FUNCTION_BLOCK OUT_ANY_TEST (* Data output to TextField *)
  (* Standard: 61499-1; Classification: GUI *)
  (* Version 0.3, 2009-02-28, JHC, Holobloc Inc, Updated service sequences. *)
  (* Version 0.2, 2009-02-23, JHC, Holobloc Inc, Updated compilers. *)
  (* Version 0.1, 2002-05-03, JHC, Rockwell Automation, Made QI IV=true. *)
  (* Version 0.0, 2001-05-31, JHC, Rockwell Automation *)
  (* Compiler header: package fb.rt.hmi; *)
  (* Compiler Java Sun JDK 1.6.0 *)
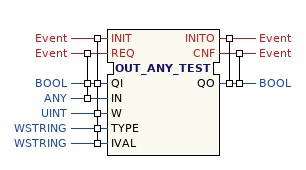
  EVENT_INPUT
    INIT WITH QI, W, TYPE, IVAL; (* Initialization *)
    REQ WITH QI, IN; (* Request *)
  END_EVENT
  EVENT_OUTPUT
    INITO WITH QO; (* Initialization Confirm *)
    CNF WITH QO; (* Service Confirmation *)
  END_EVENT
  VAR_INPUT
    QI : BOOL := true; (* Input event qualifier *)
    IN : ANY; (* Output value to convert *)
    W : UINT := 10; (* TextField width in chars *)
    TYPE : WSTRING := "ANY"; (* Data type name *)
    IVAL : WSTRING; (* Initial value *)
  END_VAR
  VAR_OUTPUT
    QO : BOOL; (* Output event qualifier *)
  END_VAR
  SERVICE Application/OUT_ANY
    SEQUENCE initialize
      Application.INIT+(LABEL) -> OUT_ANY.createTextField(W, IVAL) -> OUT_ANY.initIN(TYPE) -> Application.INITO+();
    END_SEQUENCE
    SEQUENCE field_exists
      Application.INIT+(LABEL) -> OUT_ANY.setText(IVAL) -> Application.INITO+();
    END_SEQUENCE
    SEQUENCE init_inhibited
      Application.INIT-() -> Application.INITO-();
    END_SEQUENCE
    SEQUENCE request
      Application.REQ+(LABEL) -> OUT_ANY.setText(IN.toString()) -> Application.CNF+();
    END_SEQUENCE
    SEQUENCE req_uninitialized
      Application.REQ+(LABEL) -> Application.CNF-();
    END_SEQUENCE
    SEQUENCE req_inhibited
      Application.REQ-(LABEL) -> Application.CNF-();
    END_SEQUENCE
  END_SERVICE
END_FUNCTION_BLOCK
